PROGRAM MAIN
VAR
	Machine			  : Machine := (Name := 'Machine');
	resetStateMachine : BOOL;
	abort			  : BOOL;
	stop			  : BOOL;
END_VAR

// All sample code provided by Beckhoff Automation LLC are for illustrative purposes only and are provided “as is” and without any warranties, express or implied. Actual implementations in applications will vary significantly. Beckhoff Automation LLC shall have no liability for, and does not waive any rights in relation to, any code samples that it provides or the use of such code samples for any purpose.

(*
This sample demonstrates a way to implement alarms for modules and components.
As an incorrect implementation can lead to an endless loop of Raise/CLear it is important to understand when to clear alarms.
Once of the most important details is that the _CurrentAlarmSeverity for a Component/Module must be set locally after the call to SUPER^.CyclicLogic.
This is due to the fact that _CurrentAlarmSeverity is reset to Verbose in the base class.
 

Component
	The Component includes a Monitoring method which is called by the Cyclic Logic of the base class.
	This method includes a test variable for each of the Severity levels (Verbose, Info, Warning, Error, Critical) 
	The default severities are set in the Base Class.

	Additionally, an example for changing the severity at run time is given which changes the based on the value of an pressumed Analog Input.

	Each of these Component Alarms are only cleared when the Module containing the component calls its SUPER^.Clearing()
 
Equipment Module
	The EM CyclicLogic method has code to monitor possible alarm conditions. 
	The EM does not have a Monitoring method in the base class, you can add your own and call it from CyclicLogic.
	Take note that the first 3 alarms (Verbose, Info, Warning) reset themselves once the condition is FALSE, 
	while the Error and Critical alarms are required to be reset from SUPER^.Clearing.

Machine Module
	 Most of the implementation for Alarms in the Machine module are the same as the Equipment Module.
	 The 2 differences are the implementation of a MachineMonitor, which provides similar functionality to the SubModuleMonitor method, 
	 and the way in which the Clearing method is implemented.
	 
	The MachineMonitor method is called by CyclicLogic and is a simplified version of the SubModuleMonitor in the base class,
	the SubModuleMonitor requires a FOR loop to process all of the SubModule, and this is removed from the MachineMonitor.
	
	The Clearing method is based on the one from the base class, but with the addition of a check for any Components of the Machine Module.
	More information is provided in the code.

*)

//This is for debug only and should be removed
_AppInfo.KeepOutputsOnBP := TRUE;

//
Machine.CyclicLogic();

//
CASE Machine.CurrentState OF
	E_PMLState.ePMLState_Aborted:
		IF resetStateMachine THEN
			resetStateMachine := FALSE;
			Machine.ChangeState(State := E_PMLCommand.ePMLCommand_Clear);
		END_IF

	E_PMLState.ePMLState_Stopped:
		Machine.ChangeState(State := E_PMLCommand.ePMLCommand_Reset);

	E_PMLState.ePMLState_Idle:
		Machine.ChangeState(State := E_PMLCommand.ePMLCommand_Start);
END_CASE

//
IF abort THEN
	abort := FALSE;
	Machine.ChangeState(State := E_PMLCommand.ePMLCommand_Abort);
END_IF

IF stop THEN
	stop := FALSE;
	Machine.ChangeState(State := ePMLCommand_Stop);
END_IF

END_PROGRAM

(* stored: Version 1.1.0.1, ProductVersion 3.1.4024.13
   POU MAIN: Id {31f179cd-be00-4b82-98cc-4c2f9f86690d}, SpecialFunc None *)
